// TIA Portal V16 export
// export: Created 2023-03-29T11:03:20.409134Z, ExportSetting WithDefaults, DisplayName Totally Integrated Automation Portal, DisplayVersion V16 Update 6, DisplayName TIA Portal Version Control Interface, DisplayVersion V16 Update 2, DisplayName TIA Portal Openness, DisplayVersion V16 Update 6, DisplayName STEP 7 Professional, DisplayVersion V16 Update 6, DisplayName STEP 7 Safety, DisplayVersion V16, DisplayName WinCC Advanced, DisplayVersion V16 Update 6
FUNCTION_BLOCK "WatchDog HMI"   // FB12, LAD
TITLE = WatchDog HMI
{ S7_Optimized_Access := 'TRUE' }
AUTHOR : rtecmer
VERSION : 0.1
// Kontrola komunikacji PLC z HMI. Informacja o zerwanym połączeniu przekazywana do DB SCADA WinCC
// stored: AutoNumber true, IsIECCheckEnabled false, IsRetainMemResEnabled false, MemoryReserve 500, SetENOAutomatically false, UDAEnableTagReadback false
   VAR_TEMP   // added for the SCL form of the ladder/FBD networks
      _w1 : Bool;
      _w2 : Bool;
   END_VAR
BEGIN

REGION Network 1: WatchDog HMI
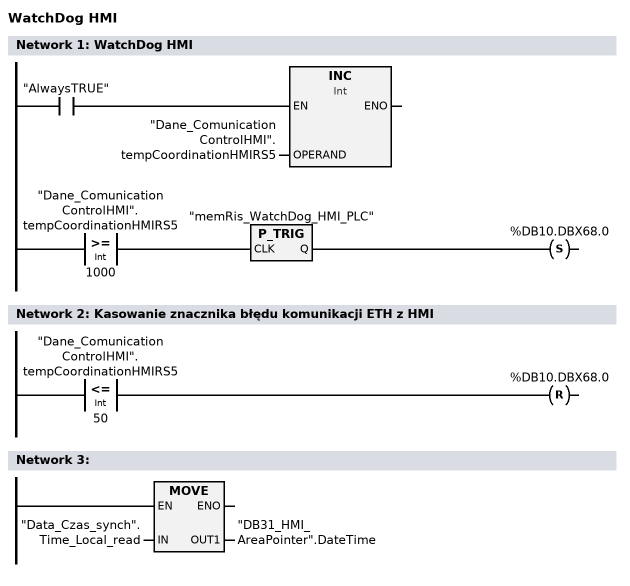
   RUNG wire#powerrail
      Contact( "AlwaysTRUE" )
      { S7_Templates := "DestType := Int" } Inc( "Dane_ComunicationControlHMI".tempCoordinationHMIRS5 )
   END_RUNG
   RUNG wire#powerrail
      { S7_Templates := "SrcType := Int" } GE_Contact(in1 := "Dane_ComunicationControlHMI".tempCoordinationHMIRS5, in2 := 1000)
      P_Trig( "memRis_WatchDog_HMI_PLC" )
      S_Coil( %DB10.DBX68.0 )
   END_RUNG
   // the same network as SCL:
   IF "AlwaysTRUE" THEN
       "Dane_ComunicationControlHMI".tempCoordinationHMIRS5 := "Dane_ComunicationControlHMI".tempCoordinationHMIRS5 + 1;
   END_IF;
   #_w1 := "Dane_ComunicationControlHMI".tempCoordinationHMIRS5 >= 1000;
   #_w2 := #_w1 AND NOT "memRis_WatchDog_HMI_PLC";   // rising edge
   "memRis_WatchDog_HMI_PLC" := #_w1;
   IF #_w2 THEN %DB10.DBX68.0 := TRUE; END_IF;
END_REGION

REGION Network 2: Kasowanie znacznika błędu komunikacji ETH z HMI
   RUNG wire#powerrail
      { S7_Templates := "SrcType := Int" } LE_Contact(in1 := "Dane_ComunicationControlHMI".tempCoordinationHMIRS5, in2 := 50)
      R_Coil( %DB10.DBX68.0 )
   END_RUNG
   // the same network as SCL:
   IF "Dane_ComunicationControlHMI".tempCoordinationHMIRS5 <= 50 THEN %DB10.DBX68.0 := FALSE; END_IF;
END_REGION

REGION Network 3
   RUNG wire#powerrail
      Move(in := "Data_Czas_synch".Time_Local_read, out1 => "DB31_HMI_AreaPointer".DateTime)
   END_RUNG
   // the same network as SCL:
   "DB31_HMI_AreaPointer".DateTime := "Data_Czas_synch".Time_Local_read;
END_REGION
END_FUNCTION_BLOCK
